(* IEC 61131-3 sources: plc_on_fpga_riscv_hybrid/RV_FPGA_PLC_IDE_Projects/And_Test, 1 file *)

(* ---- And_Test.il ---- *)
VAR
END_VAR

PROGRAM And_Test
    Rung_Number_1 :
        LD     %SW.0
        AND    %SW.1
        AND    %SW.2
        ST     %LEDG.0
END_PROGRAM
